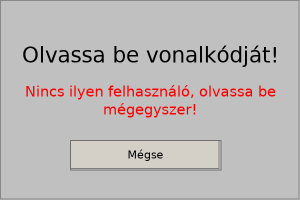
VISUALIZATION Login  // 300x200
    Label (10,40 281x30), "Olvassa be vonalkódját!"
    Button (70,140 151x30), "Mégse"
        toggle GVL.LoginEnabled
    Label (10,80 281x41), "Nincs ilyen felhasználó, olvassa be mégegyszer!", invisible if: NOT GVL.UserNotFound
END_VISUALIZATION

(* stored: Version 1.1.0.1, ProductVersion 3.1.4024.11
   Visu Login: Id {2abdd1cd-36fe-4162-a1db-cb3b731e17f0} *)
